INTERFACE ITF_BaseFlagGet

METHOD PUBLIC GetFlag : BOOL
VAR_INPUT
END_VAR
END_METHOD

END_INTERFACE

(* stored: Version 1.1.0.1
   Itf ITF_BaseFlagGet: Id {bf82d5ac-7771-0224-1c56-44ab98f3236a}
   Method GetFlag: Id {ecfd5ed9-c2f7-0d14-0ba2-89dbc527f18f} *)
